TYPE ST_BaseHMIComponent_View :
STRUCT
	wsName			: WSTRING;
	
END_STRUCT
END_TYPE

(* stored: Version 1.1.0.1
   DUT ST_BaseHMIComponent_View: Id {9a4adc48-322a-0770-2323-8e789531445d} *)
